RESOURCE_TYPE GRAPH_RESOURCE (* Resource for displaying a 3-layer (background, edges, nodes) graph *)
  (* Standard: IEC 61499; Classification: HMI; Function: Display; Type: Directed/Undirected graph *)
  (* Version 0.5, 2006-08-23, JHC, Holobloc Inc, Moved to package fb.rt.gui *)
  (* Version 0.4, 2006-08-18, JHC, Holobloc Inc, Moved all parameters to GRAPH file. *)
  (* Version 0.3, 2006-08-16, JHC, Holobloc Inc, Changed EDGES to GRAPH, deleted IMG. *)
  (* Version 0.2, 2006-08-04, JHC, Holobloc Inc, Added EDGES. *)
  (* Version 0.1, 2006-07-27, JHC, Holobloc Inc, Added FONT. *)
  (* Version 0.0, 2006-07-22, JHC, Holobloc Inc *)
  (* Compiler header: package fb.rt.gui; import java.awt.*; *)
  (* Compiler Java Sun JDK 1.5.0 *)
  VAR_INPUT
    GRAPH : WSTRING; (* Location relative to FBDK/src of XML file containing graph elements, e.g., "batch/MPP_GRAPH.xml" *)
  END_VAR
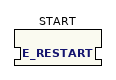
  FBS
    START : E_RESTART;
  END_FBS
END_RESOURCE_TYPE
